(********************************************************************************************************)
(*								Beckhoff Automation Poland												*)
(* 									FB_PWM_BASIC v1.1													*)
(* 										22.04.2010														*)
(*	v 1.1 - dodano bEnable, rCycleTime, początkowa faza to wyjście załączone, końcowa wyłączone			*)
(* 		Blok funkcyjny sterowania wyjsciem bOut typu BOOL na zasadzie modulowania szerokosci impulsu.	*)
(*					 Dokladnosc szerokosci impulsu  do 1 cylku sterownika.								*)
(* 							Konieczne jest dodanie biblioteki TcSystem									*)
(*______________________________________________________________________________________________________*)
FUNCTION_BLOCK FB_PWM_BASIC
VAR_INPUT
	bEnable: 			BOOL	:=TRUE;	(* Pozwolenie na działanie bloczka *)
	tPulseWidth: 		TIME; 			(*Szerokosc impulsu = 100% w ms typ zmiennej TIME*)
	fUpPercent: 		REAL; 			(*Aktualne procentowe wypelnienie impulsu*)
	rCycleTime: 		REAL;			(* Czas cylku - task, w milisekundach *)
END_VAR
VAR_OUTPUT
	bOut: 				BOOL;			(* Wyjscie *)
	wOn: 				WORD;			(* Liczba cykli z załączonym wyjściem *)
	wOff: 				WORD;			(* Liczba cykli z wyłaczonym wyjściem *)
END_VAR
VAR
	fCyclePulseWidth: 	REAL;  			(*Dlugosc impulsu = 100% w cyklach typ zmiennej REAL *)
	fCyclesOn: 			REAL;			(*Ilosc cykli, w ktorych sygnal jest zalaczony*)
	State: 				BYTE:=1;		(*Zmienna wyboru w instrukcji CASE*)
	(*Przeliczenie na pelne cykle*)
	wWidth: 			WORD;
	wCycleCounter:		WORD;			(*Licznik cykli zalaczenia/wylaczenia*)
	(*Przechowanie wartosci do porownania*)
	tPulseWidthOld: 	TIME	:= T#0MS;
	fUpPercentOld: 		REAL	:= -1;
END_VAR

IF bEnable THEN
	(*Przelicz tylko gdy zmienia sie dane*)
	IF tPulseWidth <> tPulseWidthOld OR fUpPercent <> fUpPercentOld THEN
		(*Sprawdzamy poprawnosc wprowadzonych danych*)
		IF fUpPercent <0 THEN fUpPercent := 0; END_IF
		IF fUpPercent > 100 THEN fUpPercent := 100; END_IF
		(*Obliczamy*)
		fCyclePulseWidth := TIME_TO_REAL(tPulseWidth)/rCycleTime; (*Dlugosc impulsu*)
		fCyclesOn := fCyclePulseWidth * fUpPercent/100;(*Cykle zalaczenia*)
	
		(*Przeliczamy na pelne cykle*)
		(*Opcja dla dokladniejszego przyblizenia impulsu On i Off*)
		wWidth := REAL_TO_WORD(fCyclePulseWidth);
		wOn := REAL_TO_WORD(fCyclesOn);
		(* Jeśli nie ma takiej potrzeby, nie wystawiaj wyjscia *)
		IF wOff = 0 THEN State := 0; END_IF
		wOff := REAL_TO_WORD(fCyclePulseWidth - fCyclesOn);
		(*Podstawiamy*)
		tPulseWidthOld := tPulseWidth;
		fUpPercentOld := fUpPercent;
	END_IF

	(*Albo wystawiamy TRUE albo FALSE*)
	CASE State OF
		0:
			bOut := FALSE;									(*Ustaw bOut na FALSE*)
			wCycleCounter := wCycleCounter  +  1;			(*Dodaj cykl do licznika*)
			IF wCycleCounter >= wOff THEN					(*Jezeli bylo bOut = FALSE wystarczajaca ilosc cykli to...*)
				wCycleCounter := 0;							(*Resetuj licznik*)
				IF wOff <> wWidth THEN State := 1; END_IF 	(*Przelacz tylko jesli ma byc kiedys bOut = TRUE*)
			END_IF
		1:
			bOut := TRUE;									(*Ustaw bOut na TRUE*)
			wCycleCounter := wCycleCounter  +  1;			(*Dodaj cykl do licznika*)
			IF wCycleCounter >= wOn THEN					(*Jezeli bylo bOut = TRUE wystarczajaca ilosc cykli to...*)
				wCycleCounter := 0;							(*Resetuj licznik*)
				IF wOn <> wWidth THEN State := 0; END_IF 	(*Przelacz tylko jesli ma byc kiedys bOut = FALSE*)
			END_IF
	END_CASE
ELSE
	bOut := FALSE;
	wCycleCounter := 0;
	State := 1;
END_IF

END_FUNCTION_BLOCK

(* stored: Version 1.1.0.1, ProductVersion 3.1.4026.13, FileIdentifier 026840fca88ba6c1e1261dce39c0ccc025bef1b4, FileSignature 8c4ee9f2d790f07154f220a6a50e42a7dcacae4278c4bbd913b7aad4ca3f0e36ca4997986bbc392b80f8f4164ca0dafde303e162262cee6e063b0e89e033d678d1d0271be0f49f1531c63300230edf079677c83b3902476a4d1215e15bd55859d32eb2b3439e5bcc230d03ea4f40220461b8021838147b1f78ff83c2475a09976b4d510f3e535684fa5eb82dae775c7d1423433ebf9201e64f751ed3cdbd7e08b2159f1e45892cdc924a58502b9d81964c8f99cea531f7a1226aafaa2511258c1608dcbefeec6a15efcd89075ab946d18fba69119700a9a4b9f336d4922409cc0b79b8493636eff81d97cc0fc30172fc39b43a278a19a9ab96afcdcfffbcfba9
   POU FB_PWM_BASIC: Id {cb60afbc-24ea-4917-bd4a-fcc74ed33704}, SpecialFunc None *)
